{attribute 'qualified_only'}
VAR_GLOBAL
	I AT %I* :Input;
	O AT %Q* :Output;
	Seq:FB_AutoSeq;
	Trunion:FB_Trunion;
END_VAR

(* stored: Version 1.1.0.1, ProductVersion 3.1.4024.16
   GVL Fixt2: Id {d3e95ce5-512f-46c8-9e76-6d22f630eeaa} *)
